(* IEC 61131-3 sources: s22-soft-shell/st_interpret/tests/test_inputs/st_subset_5-6, 8 files *)

(* ---- 05_And.st ---- *)
PROGRAM 05_And
    VAR
		a : bool;
		b : bool;
		c : bool;
		d : bool;
    END_VAR
		a := TRUE and False; // Result = False
		b := false & true; // Result = False
		c := False AND FALSE; // Result = False
		d := tRuE & True; // Result = True
END_PROGRAM

(* ---- 05_Or.st ---- *)
PROGRAM 05_OR
    VAR
		a : bool;
		b : bool;
		c : bool;
		d : bool;
    END_VAR
		a := TRUE or False; // Result = True
		b := false Or true; // Result = True
		c := False OR FALSE; // Result = False
		d := tRuE oR True; // Result = True
END_PROGRAM

(* ---- 05_Xor.st ---- *)
PROGRAM 05_Xor
    VAR
		a : bool;
		b : bool;
		c : bool;
		d : bool;
    END_VAR
		a := TRUE XOR False; // Result = True
		b := false xOR true; // Result = True
		c := False xOr FALSE; // Result = False
		d := tRuE xor True; // Result = False
END_PROGRAM

(* ---- 06_If.st ---- *)
//Testing simplest form of an If statement
PROGRAM 06_If
    VAR
	a : Int;
    END_VAR
    	a := 0;
        IF a < 5 THEN
		a :=  5;
        END_IF;
END_PROGRAM

(* ---- 06_If_Else.st ---- *)
//Testing simplest form of an If Else statement
PROGRAM 06_If_Else
    VAR
	a : Int;
        b : Int;
    END_VAR
	a := 0;
        b := 0;
        IF a < 5 THEN
            a :=  5;
        ELSE
            a := 3;
        END_IF;

        IF b > 5 THEN
            b :=  5;
        ELSE
            b := 3;
        END_IF;

END_PROGRAM

(* ---- 06_IF_Elsif_Else.st ---- *)
//Testing simplest form of an IF ELSIF ELSE statement
PROGRAM 07_IF_Elsif_Else
    VAR
	a : Int;
        b : Int;
        c : Int;
    END_VAR
	a := 0;
        b := 0;
        c := 0;
        IF a < 5 THEN
            a :=  5; //correct result
        ELSEIF a < 4 THEN
            a := 4;
        ELSE
            a := 3;
        END_IF;

        IF b > 5 THEN
            b :=  5;
        ELSEIF b < 4 THEN
            b := 4; //correct result
        ELSE
            b := 3;
        END_IF;

        IF c > 5 THEN
            c :=  5;
        ELSEIF c > 4 THEN
            c := 4;
        ELSE
            c := 3; //correct result
        END_IF;

END_PROGRAM

(* ---- 06_If_Nested.st ---- *)
//Testing nested form of an If statement
PROGRAM 06_If_Nested
    VAR
	a : Int;
        b : Int;
        c : Int;
    END_VAR
	a := 0;
        b := 0;
        c := 0;
        IF a < 5 THEN
            a :=  5;
            IF b < 5 THEN
                b :=  4;
                IF c < 5 THEN
                    c :=  3;
                END_IF;
            END_IF;
            IF c < 1 THEN
                    c :=  5;
            END_IF;
        END_IF;
END_PROGRAM

(* ---- 06_Not.st ---- *)
PROGRAM 05_Not
    VAR
		a : bool;
		b : bool;
    END_VAR
		a := not false; // Result = True
		b := NOT true; // Result = False
END_PROGRAM
